// TIA Portal project "plc_industrial_sorter" (V17)

(* hardware
DEVICE "S7-1500/ET200MP station_1"  S7-1500 station
   slot 0: "Rail_0"  Rack  6ES7 590-1***0-0AA0
   slot 1: "PLC_1"  CPU 1511-1 PN  6ES7 511-1AK00-0AB0  V1.8
      slot 3: "CPU display_1"  6ES7591-1AA00-0AA0
      slot 32768: "PROFINET interface_1"  X1
         slot 32769: "Port_1"  X1 P1
         slot 32770: "Port_2"  X1 P2
*)

// ===== PLC "PLC_1"  CPU 1511-1 PN =====

DATA_BLOCK "Data_block_1"   // DB1
{ S7_Optimized_Access := 'TRUE' }
VERSION : 0.1
   VAR
      Nastro1_run : Bool;
      Fotocellula_ingresso_nastro1 : Bool;
      Val_induttivo : Bool;
      Val_capacitivo : Bool;
      Peso : Real;
      Fotocellula_scan : Bool;
      Fotocellula_ingresso_nastro2 : Bool;
      Tip_oggetto : Int := 0;
      Nastro2_run : Bool;
      Pusher_avanza : Bool;
      Pusher_rientra : Bool;
      Posizione_carrello : Int;
      State_machine : Int;
      Contenitore_target : Int;
      Posizione_target_carrello : Int;
      Posizione_oggetto_Y : Real;
      Posizione_oggetto_X : Real := -1000.0;
      Sistema_START : Bool;
      Sistema_STOP : Bool;
      Sistema_ANNULLA_ALLARMI : Bool;
      Sistema_avviato : Bool;
      tempvar1 : Int;
      Contatore : Int := -1;
      Allarme_generale : Bool;
   END_VAR
BEGIN
END_DATA_BLOCK

// folder: System blocks/Program resources

DATA_BLOCK "IEC_Timer_0_DB_2"   // DB4
{ S7_Optimized_Access := 'TRUE' }
AUTHOR : Simatic
FAMILY : IEC
NAME : IEC_TMR
VERSION : 1.0
// stored: InstanceOfName IEC_TIMER
"IEC_TIMER"
BEGIN
END_DATA_BLOCK

DATA_BLOCK "IEC_Timer_0_DB_1X"   // DB6
{ S7_Optimized_Access := 'TRUE' }
AUTHOR : Simatic
FAMILY : IEC
NAME : IEC_TMR
VERSION : 1.0
// stored: InstanceOfName IEC_TIMER
"IEC_TIMER"
BEGIN
END_DATA_BLOCK

DATA_BLOCK "IEC_Timer_0_DB_6"   // DB12
{ S7_Optimized_Access := 'TRUE' }
AUTHOR : Simatic
FAMILY : IEC
NAME : IEC_TMR
VERSION : 1.0
// stored: InstanceOfName IEC_TIMER
"IEC_TIMER"
BEGIN
END_DATA_BLOCK

DATA_BLOCK "IEC_Timer_0_DB_7"   // DB13
{ S7_Optimized_Access := 'TRUE' }
AUTHOR : Simatic
FAMILY : IEC
NAME : IEC_TMR
VERSION : 1.0
// stored: InstanceOfName IEC_TIMER
"IEC_TIMER"
BEGIN
END_DATA_BLOCK

DATA_BLOCK "IEC_Timer_0_DB_8"   // DB14
{ S7_Optimized_Access := 'TRUE' }
AUTHOR : Simatic
FAMILY : IEC
NAME : IEC_TMR
VERSION : 1.0
// stored: InstanceOfName IEC_TIMER
"IEC_TIMER"
BEGIN
END_DATA_BLOCK

DATA_BLOCK "IEC_Timer_0_DB_10"   // DB16
{ S7_Optimized_Access := 'TRUE' }
AUTHOR : Simatic
FAMILY : IEC
NAME : IEC_TMR
VERSION : 1.0
// stored: InstanceOfName IEC_TIMER
"IEC_TIMER"
BEGIN
END_DATA_BLOCK

DATA_BLOCK "IEC_Timer_0_DB_11"   // DB17
{ S7_Optimized_Access := 'TRUE' }
AUTHOR : Simatic
FAMILY : IEC
NAME : IEC_TMR
VERSION : 1.0
// stored: InstanceOfName IEC_TIMER
"IEC_TIMER"
BEGIN
END_DATA_BLOCK

DATA_BLOCK "IEC_Timer_0_DB_12"   // DB18
{ S7_Optimized_Access := 'TRUE' }
AUTHOR : Simatic
FAMILY : IEC
NAME : IEC_TMR
VERSION : 1.0
// stored: InstanceOfName IEC_TIMER
"IEC_TIMER"
BEGIN
END_DATA_BLOCK

// folder: (top level)

ORGANIZATION_BLOCK "Main"   // OB1, LAD, ProgramCycle
TITLE = "Main Program Sweep (Cycle)"
{ S7_Optimized_Access := 'TRUE' }
VERSION : 0.1
   VAR_INPUT
      Initial_Call : Bool;   // Initial call of this OB
      Remanence : Bool;   // =True, if remanent data are available
   END_VAR
   VAR_TEMP   // added for the SCL form of the ladder/FBD networks
      _w1 : Bool;
      _w2 : Bool;
   END_VAR
BEGIN

REGION Network 1
   // settato il blocco totale del sistema
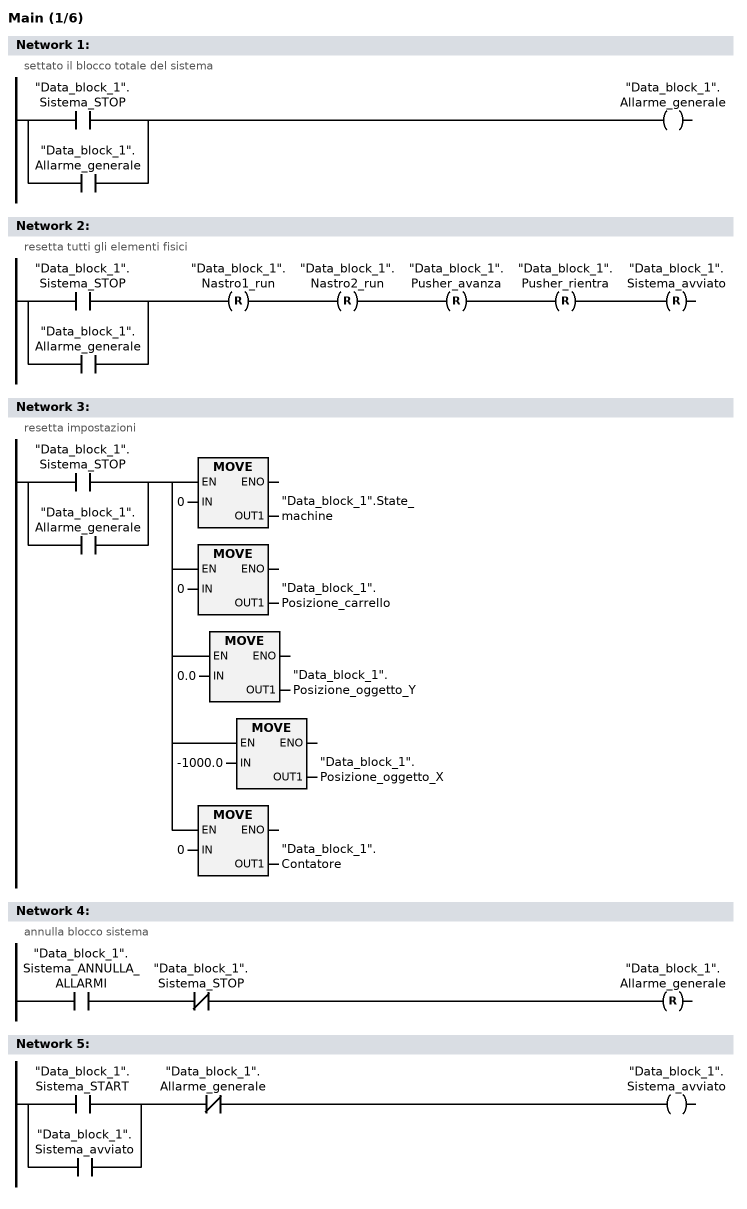
   RUNG wire#powerrail
      Contact( "Data_block_1".Sistema_STOP )
      wire#w1
      Coil( "Data_block_1".Allarme_generale )
   END_RUNG
   RUNG wire#powerrail
      Contact( "Data_block_1".Allarme_generale )
   END_RUNG wire#w1
   // the same network as SCL:
   "Data_block_1".Allarme_generale := "Data_block_1".Sistema_STOP OR "Data_block_1".Allarme_generale;
END_REGION

REGION Network 2
   // resetta tutti gli elementi fisici
   RUNG wire#powerrail
      Contact( "Data_block_1".Sistema_STOP )
      wire#w1
      R_Coil( "Data_block_1".Nastro1_run )
      R_Coil( "Data_block_1".Nastro2_run )
      R_Coil( "Data_block_1".Pusher_avanza )
      R_Coil( "Data_block_1".Pusher_rientra )
      R_Coil( "Data_block_1".Sistema_avviato )
   END_RUNG
   RUNG wire#powerrail
      Contact( "Data_block_1".Allarme_generale )
   END_RUNG wire#w1
   // the same network as SCL:
   IF "Data_block_1".Sistema_STOP OR "Data_block_1".Allarme_generale THEN
       "Data_block_1".Nastro1_run := FALSE;
       "Data_block_1".Nastro2_run := FALSE;
       "Data_block_1".Pusher_avanza := FALSE;
       "Data_block_1".Pusher_rientra := FALSE;
       "Data_block_1".Sistema_avviato := FALSE;
   END_IF;
END_REGION

REGION Network 3
   // resetta impostazioni
   RUNG wire#powerrail
      Contact( "Data_block_1".Sistema_STOP )
      wire#w1
      Move(in := 0, out1 => "Data_block_1".State_machine)
   END_RUNG
   RUNG wire#powerrail
      Contact( "Data_block_1".Allarme_generale )
   END_RUNG wire#w1
   RUNG wire#w1
      Move(in := 0, out1 => "Data_block_1".Posizione_carrello)
   END_RUNG
   RUNG wire#w1
      Move(in := 0.0, out1 => "Data_block_1".Posizione_oggetto_Y)
   END_RUNG
   RUNG wire#w1
      Move(in := -1000.0, out1 => "Data_block_1".Posizione_oggetto_X)
   END_RUNG
   RUNG wire#w1
      Move(in := 0, out1 => "Data_block_1".Contatore)
   END_RUNG
   // the same network as SCL:
   IF "Data_block_1".Sistema_STOP OR "Data_block_1".Allarme_generale THEN
       "Data_block_1".State_machine := 0;
       "Data_block_1".Posizione_carrello := 0;
       "Data_block_1".Posizione_oggetto_Y := 0.0;
       "Data_block_1".Posizione_oggetto_X := -1000.0;
       "Data_block_1".Contatore := 0;
   END_IF;
END_REGION

REGION Network 4
   // annulla blocco sistema
   RUNG wire#powerrail
      Contact( "Data_block_1".Sistema_ANNULLA_ALLARMI )
      I_Contact( "Data_block_1".Sistema_STOP )
      R_Coil( "Data_block_1".Allarme_generale )
   END_RUNG
   // the same network as SCL:
   IF "Data_block_1".Sistema_ANNULLA_ALLARMI AND NOT "Data_block_1".Sistema_STOP THEN
       "Data_block_1".Allarme_generale := FALSE;
   END_IF;
END_REGION

REGION Network 5
   RUNG wire#powerrail
      Contact( "Data_block_1".Sistema_START )
      wire#w1
      I_Contact( "Data_block_1".Allarme_generale )
      Coil( "Data_block_1".Sistema_avviato )
   END_RUNG
   RUNG wire#powerrail
      Contact( "Data_block_1".Sistema_avviato )
   END_RUNG wire#w1
   // the same network as SCL:
   "Data_block_1".Sistema_avviato := ("Data_block_1".Sistema_START OR "Data_block_1".Sistema_avviato) AND NOT "Data_block_1".Allarme_generale;
END_REGION

REGION Network 6
   // rung supporto (inizializza la fotocellula primo avvio)
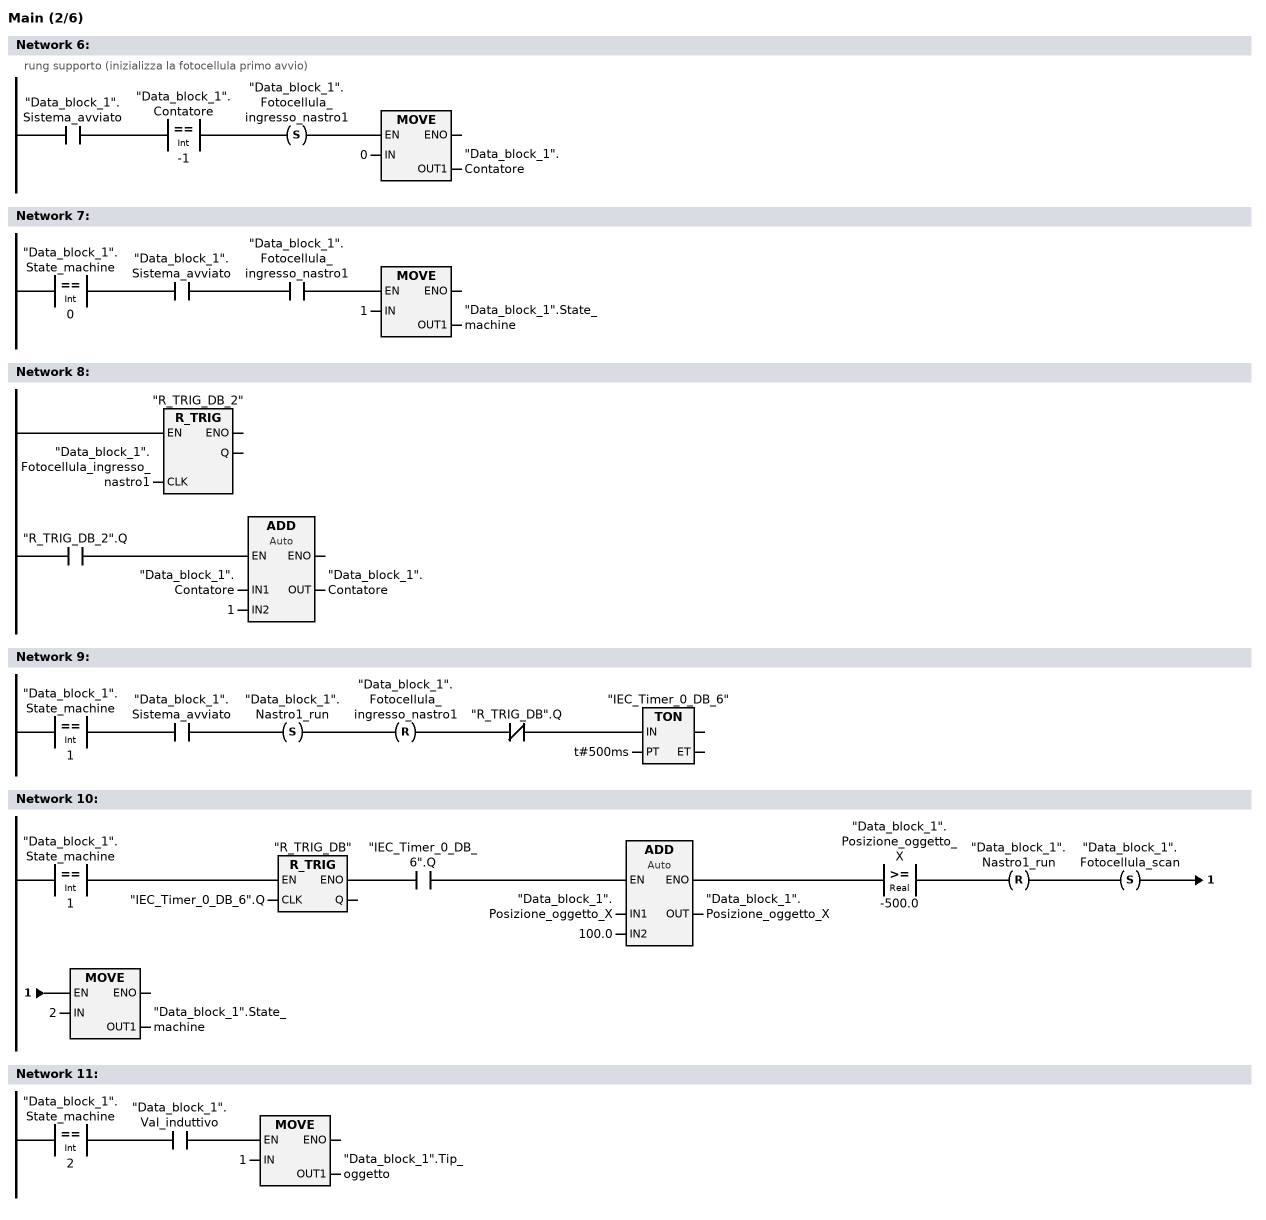
   RUNG wire#powerrail
      Contact( "Data_block_1".Sistema_avviato )
      { S7_Templates := "SrcType := Int" } EQ_Contact(in1 := "Data_block_1".Contatore, in2 := -1)
      S_Coil( "Data_block_1".Fotocellula_ingresso_nastro1 )
      Move(in := 0, out1 => "Data_block_1".Contatore)
   END_RUNG
   // the same network as SCL:
   IF "Data_block_1".Sistema_avviato AND ("Data_block_1".Contatore = (-1)) THEN
       "Data_block_1".Fotocellula_ingresso_nastro1 := TRUE;
       "Data_block_1".Contatore := 0;
   END_IF;
END_REGION

REGION Network 7
   RUNG wire#powerrail
      { S7_Templates := "SrcType := Int" } EQ_Contact(in1 := "Data_block_1".State_machine, in2 := 0)
      Contact( "Data_block_1".Sistema_avviato )
      Contact( "Data_block_1".Fotocellula_ingresso_nastro1 )
      Move(in := 1, out1 => "Data_block_1".State_machine)
   END_RUNG
   // the same network as SCL:
   IF ("Data_block_1".State_machine = 0) AND "Data_block_1".Sistema_avviato AND "Data_block_1".Fotocellula_ingresso_nastro1 THEN
       "Data_block_1".State_machine := 1;
   END_IF;
END_REGION

REGION Network 8
   "R_TRIG_DB_2"(CLK := "Data_block_1".Fotocellula_ingresso_nastro1);   // R_TRIG
   IF "R_TRIG_DB_2".Q THEN "Data_block_1".Contatore := "Data_block_1".Contatore + 1; END_IF;
END_REGION

REGION Network 9
   #_w1 := ("Data_block_1".State_machine = 1) AND "Data_block_1".Sistema_avviato;
   IF #_w1 THEN
       "Data_block_1".Nastro1_run := TRUE;
       "Data_block_1".Fotocellula_ingresso_nastro1 := FALSE;
   END_IF;
   "IEC_Timer_0_DB_6".TON(IN := #_w1 AND NOT "R_TRIG_DB".Q, PT := t#500ms);
END_REGION

REGION Network 10
   // ENO of a box is taken as its EN; it also drops when the box reports an error
   #_w1 := "Data_block_1".State_machine = 1;
   IF #_w1 THEN
       "R_TRIG_DB"(CLK := "IEC_Timer_0_DB_6".Q);   // R_TRIG
   END_IF;
   #_w2 := #_w1 AND "IEC_Timer_0_DB_6".Q;
   IF #_w2 THEN "Data_block_1".Posizione_oggetto_X := "Data_block_1".Posizione_oggetto_X + 100.0; END_IF;
   IF #_w2 AND ("Data_block_1".Posizione_oggetto_X >= (-500.0)) THEN
       "Data_block_1".Nastro1_run := FALSE;
       "Data_block_1".Fotocellula_scan := TRUE;
       "Data_block_1".State_machine := 2;
   END_IF;
END_REGION

REGION Network 11
   RUNG wire#powerrail
      { S7_Templates := "SrcType := Int" } EQ_Contact(in1 := "Data_block_1".State_machine, in2 := 2)
      Contact( "Data_block_1".Val_induttivo )
      Move(in := 1, out1 => "Data_block_1".Tip_oggetto)
   END_RUNG
   // the same network as SCL:
   IF ("Data_block_1".State_machine = 2) AND "Data_block_1".Val_induttivo THEN
       "Data_block_1".Tip_oggetto := 1;
   END_IF;
END_REGION

REGION Network 12
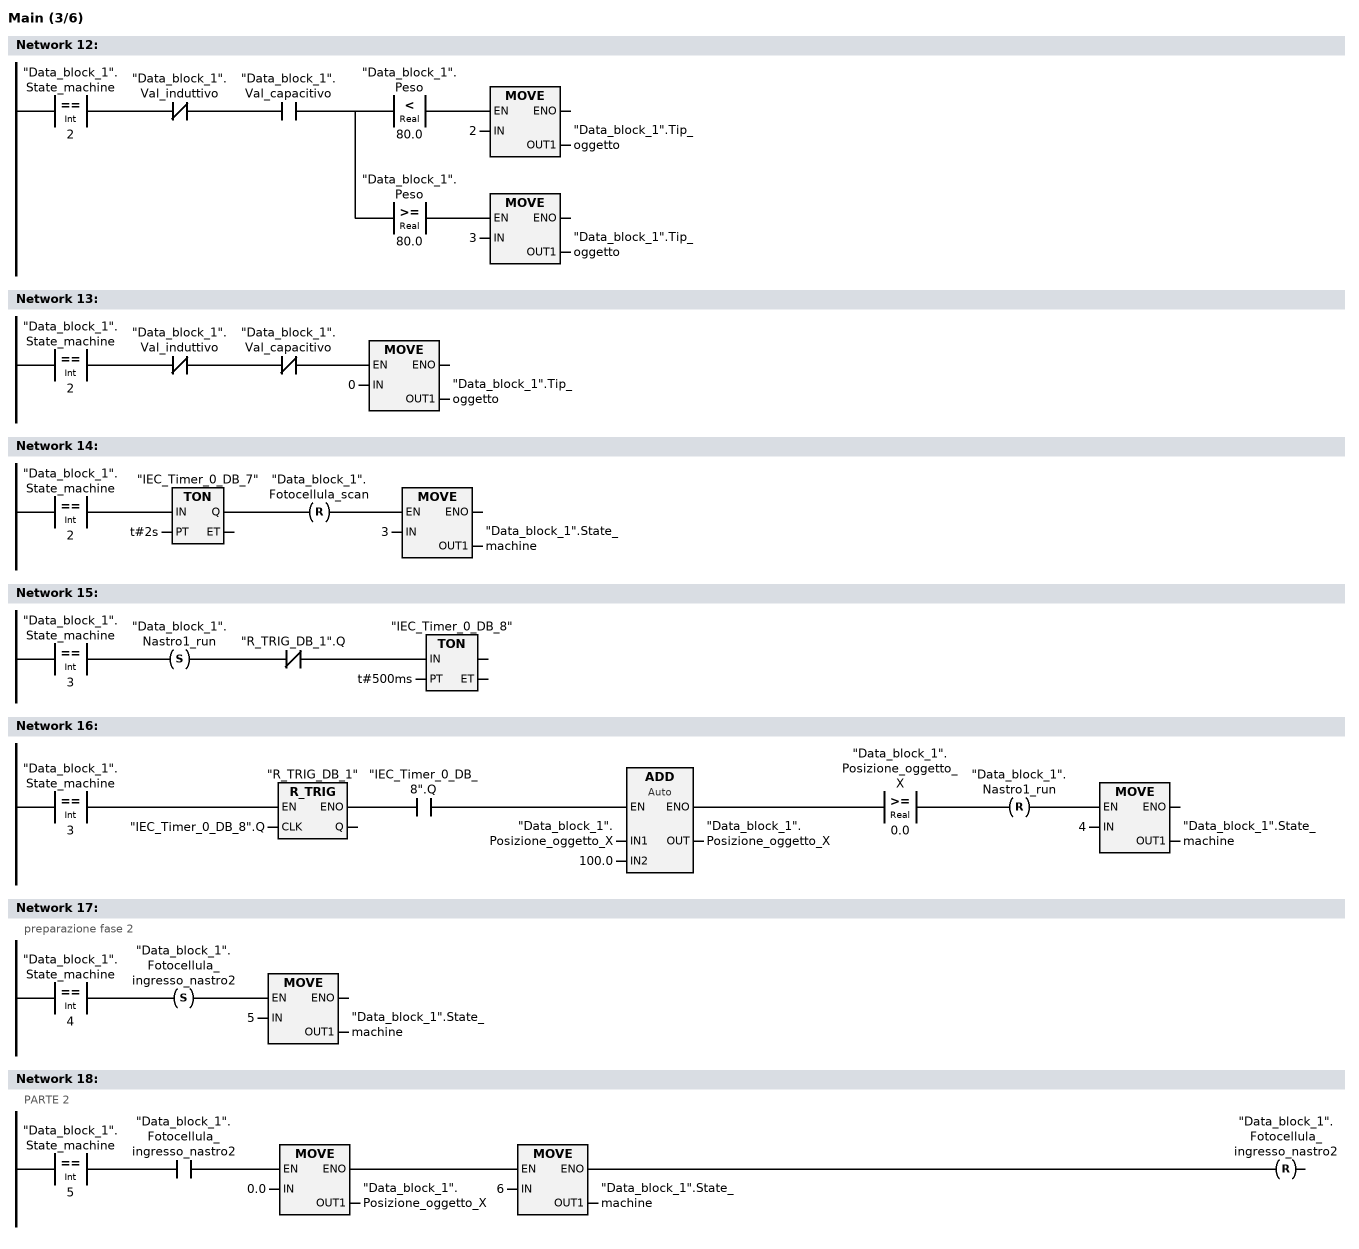
   RUNG wire#powerrail
      { S7_Templates := "SrcType := Int" } EQ_Contact(in1 := "Data_block_1".State_machine, in2 := 2)
      I_Contact( "Data_block_1".Val_induttivo )
      Contact( "Data_block_1".Val_capacitivo )
      wire#w1
      { S7_Templates := "SrcType := Real" } LT_Contact(in1 := "Data_block_1".Peso, in2 := 80.0)
      Move(in := 2, out1 => "Data_block_1".Tip_oggetto)
   END_RUNG
   RUNG wire#w1
      { S7_Templates := "SrcType := Real" } GE_Contact(in1 := "Data_block_1".Peso, in2 := 80.0)
      Move(in := 3, out1 => "Data_block_1".Tip_oggetto)
   END_RUNG
   // the same network as SCL:
   #_w1 := ("Data_block_1".State_machine = 2) AND NOT "Data_block_1".Val_induttivo AND "Data_block_1".Val_capacitivo;
   IF #_w1 AND ("Data_block_1".Peso < 80.0) THEN "Data_block_1".Tip_oggetto := 2; END_IF;
   IF #_w1 AND ("Data_block_1".Peso >= 80.0) THEN "Data_block_1".Tip_oggetto := 3; END_IF;
END_REGION

REGION Network 13
   RUNG wire#powerrail
      { S7_Templates := "SrcType := Int" } EQ_Contact(in1 := "Data_block_1".State_machine, in2 := 2)
      I_Contact( "Data_block_1".Val_induttivo )
      I_Contact( "Data_block_1".Val_capacitivo )
      Move(in := 0, out1 => "Data_block_1".Tip_oggetto)
   END_RUNG
   // the same network as SCL:
   IF ("Data_block_1".State_machine = 2) AND NOT "Data_block_1".Val_induttivo AND NOT "Data_block_1".Val_capacitivo THEN
       "Data_block_1".Tip_oggetto := 0;
   END_IF;
END_REGION

REGION Network 14
   "IEC_Timer_0_DB_7".TON(IN := "Data_block_1".State_machine = 2, PT := t#2s);
   IF "IEC_Timer_0_DB_7".Q THEN
       "Data_block_1".Fotocellula_scan := FALSE;
       "Data_block_1".State_machine := 3;
   END_IF;
END_REGION

REGION Network 15
   #_w1 := "Data_block_1".State_machine = 3;
   IF #_w1 THEN "Data_block_1".Nastro1_run := TRUE; END_IF;
   "IEC_Timer_0_DB_8".TON(IN := #_w1 AND NOT "R_TRIG_DB_1".Q, PT := t#500ms);
END_REGION

REGION Network 16
   // ENO of a box is taken as its EN; it also drops when the box reports an error
   #_w1 := "Data_block_1".State_machine = 3;
   IF #_w1 THEN
       "R_TRIG_DB_1"(CLK := "IEC_Timer_0_DB_8".Q);   // R_TRIG
   END_IF;
   #_w2 := #_w1 AND "IEC_Timer_0_DB_8".Q;
   IF #_w2 THEN "Data_block_1".Posizione_oggetto_X := "Data_block_1".Posizione_oggetto_X + 100.0; END_IF;
   IF #_w2 AND ("Data_block_1".Posizione_oggetto_X >= 0.0) THEN
       "Data_block_1".Nastro1_run := FALSE;
       "Data_block_1".State_machine := 4;
   END_IF;
END_REGION

REGION Network 17
   // preparazione fase 2
   RUNG wire#powerrail
      { S7_Templates := "SrcType := Int" } EQ_Contact(in1 := "Data_block_1".State_machine, in2 := 4)
      S_Coil( "Data_block_1".Fotocellula_ingresso_nastro2 )
      Move(in := 5, out1 => "Data_block_1".State_machine)
   END_RUNG
   // the same network as SCL:
   IF "Data_block_1".State_machine = 4 THEN
       "Data_block_1".Fotocellula_ingresso_nastro2 := TRUE;
       "Data_block_1".State_machine := 5;
   END_IF;
END_REGION

REGION Network 18
   // PARTE 2
   RUNG wire#powerrail
      { S7_Templates := "SrcType := Int" } EQ_Contact(in1 := "Data_block_1".State_machine, in2 := 5)
      Contact( "Data_block_1".Fotocellula_ingresso_nastro2 )
      Move(in := 0.0, out1 => "Data_block_1".Posizione_oggetto_X)
      Move(in := 6, out1 => "Data_block_1".State_machine)
      R_Coil( "Data_block_1".Fotocellula_ingresso_nastro2 )
   END_RUNG
   // the same network as SCL:
   IF ("Data_block_1".State_machine = 5) AND "Data_block_1".Fotocellula_ingresso_nastro2 THEN
       "Data_block_1".Posizione_oggetto_X := 0.0;
   END_IF;
   #_w1 := ("Data_block_1".State_machine = 5) AND "Data_block_1".Fotocellula_ingresso_nastro2;
   IF #_w1 THEN
       "Data_block_1".State_machine := 6;
       "Data_block_1".Fotocellula_ingresso_nastro2 := FALSE;
   END_IF;
END_REGION

REGION Network 19
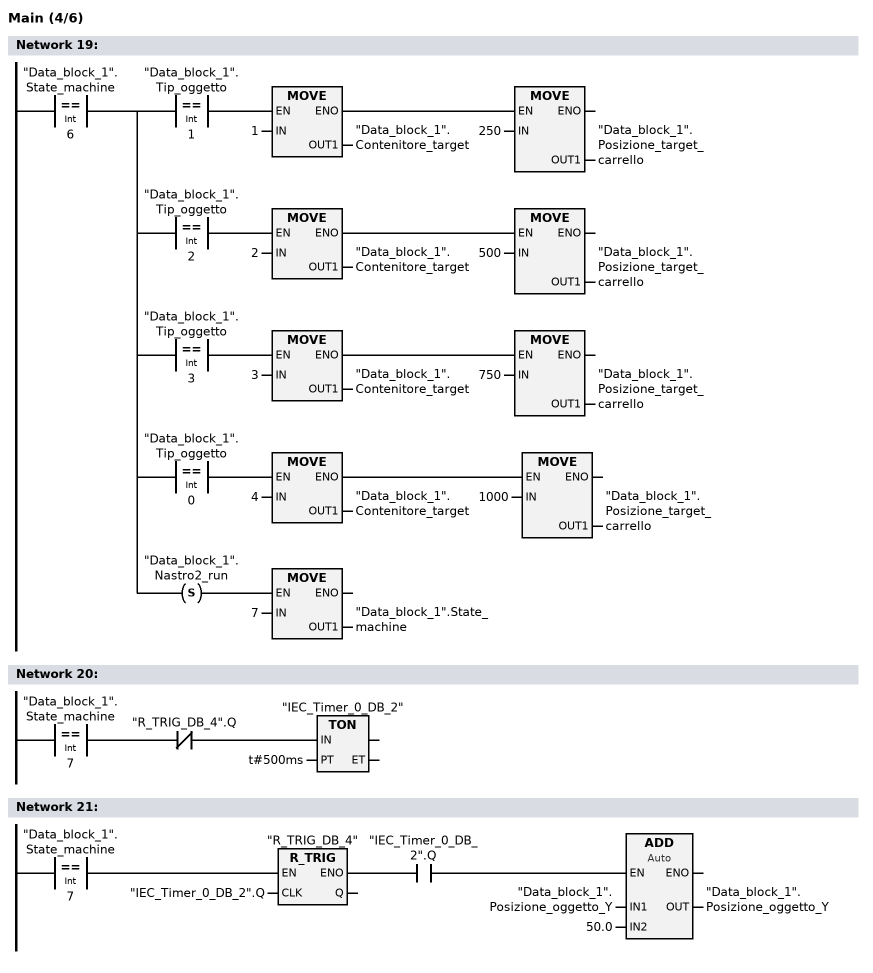
   RUNG wire#powerrail
      { S7_Templates := "SrcType := Int" } EQ_Contact(in1 := "Data_block_1".State_machine, in2 := 6)
      wire#w1
      { S7_Templates := "SrcType := Int" } EQ_Contact(in1 := "Data_block_1".Tip_oggetto, in2 := 1)
      Move(in := 1, out1 => "Data_block_1".Contenitore_target)
      Move(in := 250, out1 => "Data_block_1".Posizione_target_carrello)
   END_RUNG
   RUNG wire#w1
      { S7_Templates := "SrcType := Int" } EQ_Contact(in1 := "Data_block_1".Tip_oggetto, in2 := 2)
      Move(in := 2, out1 => "Data_block_1".Contenitore_target)
      Move(in := 500, out1 => "Data_block_1".Posizione_target_carrello)
   END_RUNG
   RUNG wire#w1
      { S7_Templates := "SrcType := Int" } EQ_Contact(in1 := "Data_block_1".Tip_oggetto, in2 := 3)
      Move(in := 3, out1 => "Data_block_1".Contenitore_target)
      Move(in := 750, out1 => "Data_block_1".Posizione_target_carrello)
   END_RUNG
   RUNG wire#w1
      { S7_Templates := "SrcType := Int" } EQ_Contact(in1 := "Data_block_1".Tip_oggetto, in2 := 0)
      Move(in := 4, out1 => "Data_block_1".Contenitore_target)
      Move(in := 1000, out1 => "Data_block_1".Posizione_target_carrello)
   END_RUNG
   RUNG wire#w1
      S_Coil( "Data_block_1".Nastro2_run )
      Move(in := 7, out1 => "Data_block_1".State_machine)
   END_RUNG
   // the same network as SCL:
   #_w1 := "Data_block_1".State_machine = 6;
   IF #_w1 AND ("Data_block_1".Tip_oggetto = 1) THEN
       "Data_block_1".Contenitore_target := 1;
       "Data_block_1".Posizione_target_carrello := 250;
   END_IF;
   IF #_w1 AND ("Data_block_1".Tip_oggetto = 2) THEN
       "Data_block_1".Contenitore_target := 2;
       "Data_block_1".Posizione_target_carrello := 500;
   END_IF;
   IF #_w1 AND ("Data_block_1".Tip_oggetto = 3) THEN
       "Data_block_1".Contenitore_target := 3;
       "Data_block_1".Posizione_target_carrello := 750;
   END_IF;
   IF #_w1 AND ("Data_block_1".Tip_oggetto = 0) THEN
       "Data_block_1".Contenitore_target := 4;
       "Data_block_1".Posizione_target_carrello := 1000;
   END_IF;
   IF #_w1 THEN
       "Data_block_1".Nastro2_run := TRUE;
       "Data_block_1".State_machine := 7;
   END_IF;
END_REGION

REGION Network 20
   "IEC_Timer_0_DB_2".TON(IN := ("Data_block_1".State_machine = 7) AND NOT "R_TRIG_DB_4".Q, PT := t#500ms);
END_REGION

REGION Network 21
   // ENO of a box is taken as its EN; it also drops when the box reports an error
   #_w1 := "Data_block_1".State_machine = 7;
   IF #_w1 THEN
       "R_TRIG_DB_4"(CLK := "IEC_Timer_0_DB_2".Q);   // R_TRIG
   END_IF;
   IF #_w1 AND "IEC_Timer_0_DB_2".Q THEN
       "Data_block_1".Posizione_oggetto_Y := "Data_block_1".Posizione_oggetto_Y + 50.0;
   END_IF;
END_REGION

REGION Network 22
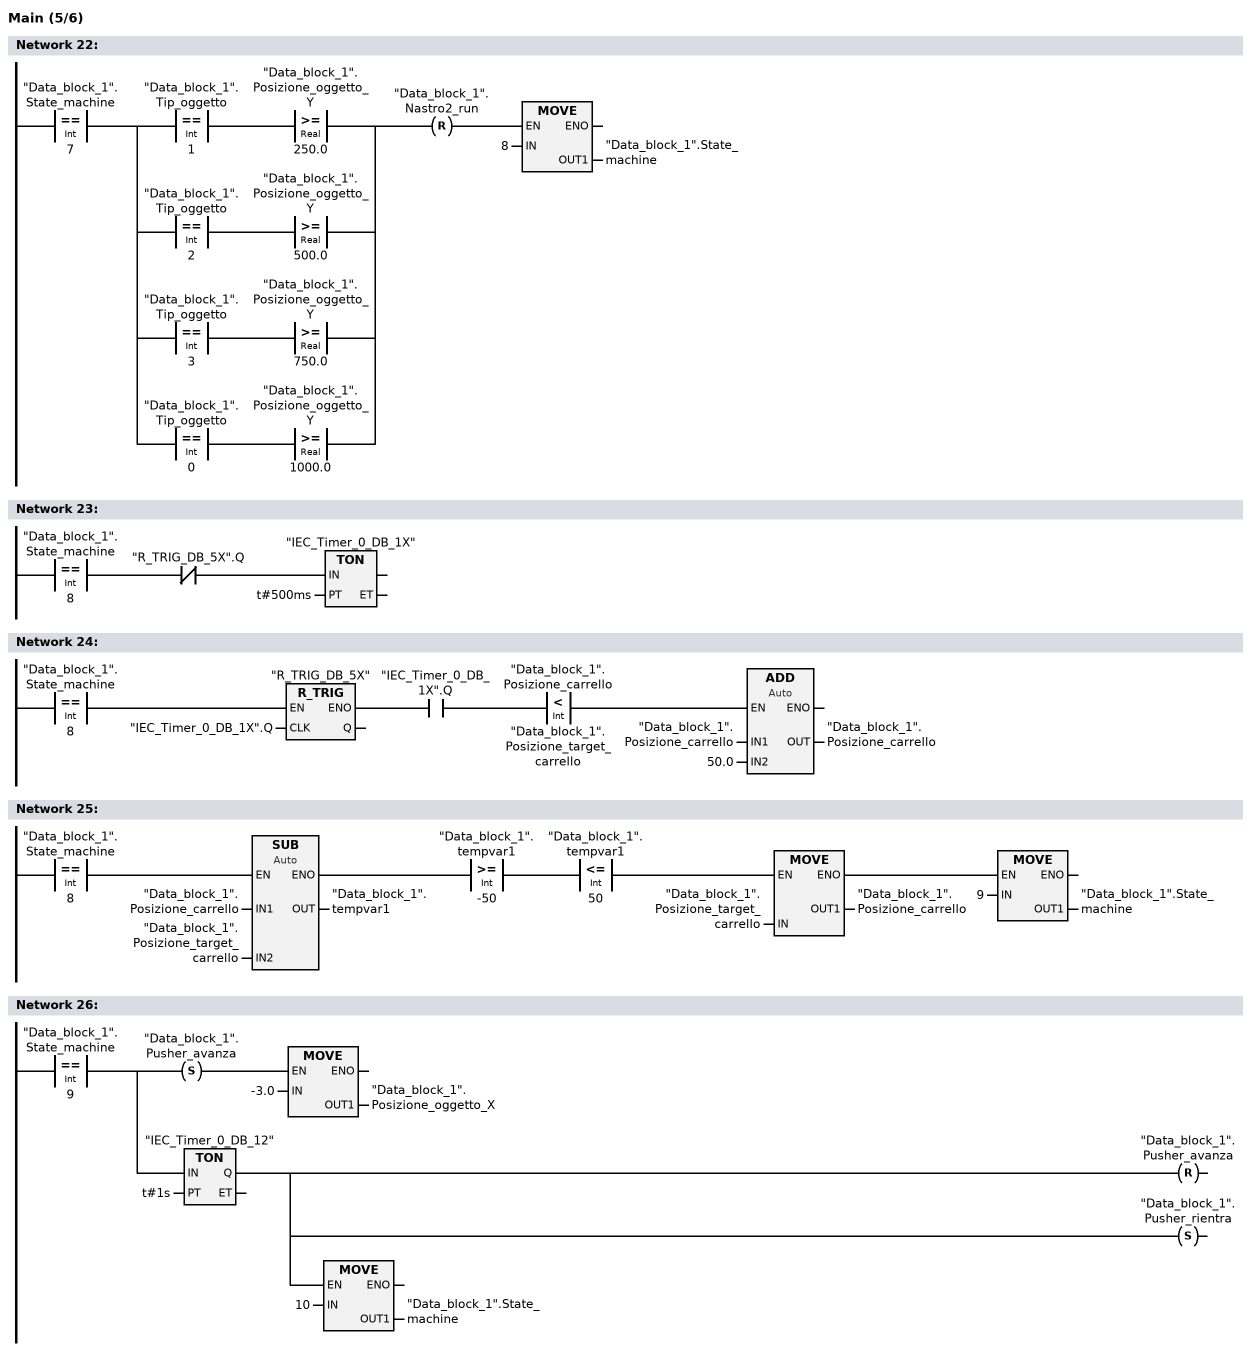
   RUNG wire#powerrail
      { S7_Templates := "SrcType := Int" } EQ_Contact(in1 := "Data_block_1".State_machine, in2 := 7)
      wire#w1
      { S7_Templates := "SrcType := Int" } EQ_Contact(in1 := "Data_block_1".Tip_oggetto, in2 := 1)
      { S7_Templates := "SrcType := Real" } GE_Contact(in1 := "Data_block_1".Posizione_oggetto_Y, in2 := 250.0)
      wire#w2
      R_Coil( "Data_block_1".Nastro2_run )
      Move(in := 8, out1 => "Data_block_1".State_machine)
   END_RUNG
   RUNG wire#w1
      { S7_Templates := "SrcType := Int" } EQ_Contact(in1 := "Data_block_1".Tip_oggetto, in2 := 2)
      { S7_Templates := "SrcType := Real" } GE_Contact(in1 := "Data_block_1".Posizione_oggetto_Y, in2 := 500.0)
   END_RUNG wire#w2
   RUNG wire#w1
      { S7_Templates := "SrcType := Int" } EQ_Contact(in1 := "Data_block_1".Tip_oggetto, in2 := 3)
      { S7_Templates := "SrcType := Real" } GE_Contact(in1 := "Data_block_1".Posizione_oggetto_Y, in2 := 750.0)
   END_RUNG wire#w2
   RUNG wire#w1
      { S7_Templates := "SrcType := Int" } EQ_Contact(in1 := "Data_block_1".Tip_oggetto, in2 := 0)
      { S7_Templates := "SrcType := Real" } GE_Contact(in1 := "Data_block_1".Posizione_oggetto_Y, in2 := 1000.0)
   END_RUNG wire#w2
   // the same network as SCL:
   IF ("Data_block_1".State_machine = 7) AND ((("Data_block_1".Tip_oggetto = 1) AND ("Data_block_1".Posizione_oggetto_Y >= 250.0)) OR (("Data_block_1".Tip_oggetto = 2) AND ("Data_block_1".Posizione_oggetto_Y >= 500.0)) OR (("Data_block_1".Tip_oggetto = 3) AND ("Data_block_1".Posizione_oggetto_Y >= 750.0)) OR (("Data_block_1".Tip_oggetto = 0) AND ("Data_block_1".Posizione_oggetto_Y >= 1000.0))) THEN
       "Data_block_1".Nastro2_run := FALSE;
       "Data_block_1".State_machine := 8;
   END_IF;
END_REGION

REGION Network 23
   "IEC_Timer_0_DB_1X".TON(IN := ("Data_block_1".State_machine = 8) AND NOT "R_TRIG_DB_5X".Q, PT := t#500ms);
END_REGION

REGION Network 24
   // ENO of a box is taken as its EN; it also drops when the box reports an error
   #_w1 := "Data_block_1".State_machine = 8;
   IF #_w1 THEN
       "R_TRIG_DB_5X"(CLK := "IEC_Timer_0_DB_1X".Q);   // R_TRIG
   END_IF;
   IF #_w1 AND "IEC_Timer_0_DB_1X".Q AND ("Data_block_1".Posizione_carrello < "Data_block_1".Posizione_target_carrello) THEN
       "Data_block_1".Posizione_carrello := "Data_block_1".Posizione_carrello + 50.0;
   END_IF;
END_REGION

REGION Network 25
   RUNG wire#powerrail
      { S7_Templates := "SrcType := Int" } EQ_Contact(in1 := "Data_block_1".State_machine, in2 := 8)
      Sub(in1 := "Data_block_1".Posizione_carrello, in2 := "Data_block_1".Posizione_target_carrello, out => "Data_block_1".tempvar1)
      { S7_Templates := "SrcType := Int" } GE_Contact(in1 := "Data_block_1".tempvar1, in2 := -50)
      { S7_Templates := "SrcType := Int" } LE_Contact(in1 := "Data_block_1".tempvar1, in2 := 50)
      Move(in := "Data_block_1".Posizione_target_carrello, out1 => "Data_block_1".Posizione_carrello)
      Move(in := 9, out1 => "Data_block_1".State_machine)
   END_RUNG
   // the same network as SCL:
   #_w1 := "Data_block_1".State_machine = 8;
   IF #_w1 THEN
       "Data_block_1".tempvar1 := "Data_block_1".Posizione_carrello - "Data_block_1".Posizione_target_carrello;
   END_IF;
   IF #_w1 AND ("Data_block_1".tempvar1 >= (-50)) AND ("Data_block_1".tempvar1 <= 50) THEN
       "Data_block_1".Posizione_carrello := "Data_block_1".Posizione_target_carrello;
       "Data_block_1".State_machine := 9;
   END_IF;
END_REGION

REGION Network 26
   #_w1 := "Data_block_1".State_machine = 9;
   IF #_w1 THEN
       "Data_block_1".Pusher_avanza := TRUE;
       "Data_block_1".Posizione_oggetto_X := -3.0;
   END_IF;
   "IEC_Timer_0_DB_12".TON(IN := #_w1, PT := t#1s);
   IF "IEC_Timer_0_DB_12".Q THEN
       "Data_block_1".Pusher_avanza := FALSE;
       "Data_block_1".Pusher_rientra := TRUE;
       "Data_block_1".State_machine := 10;
   END_IF;
END_REGION

REGION Network 27
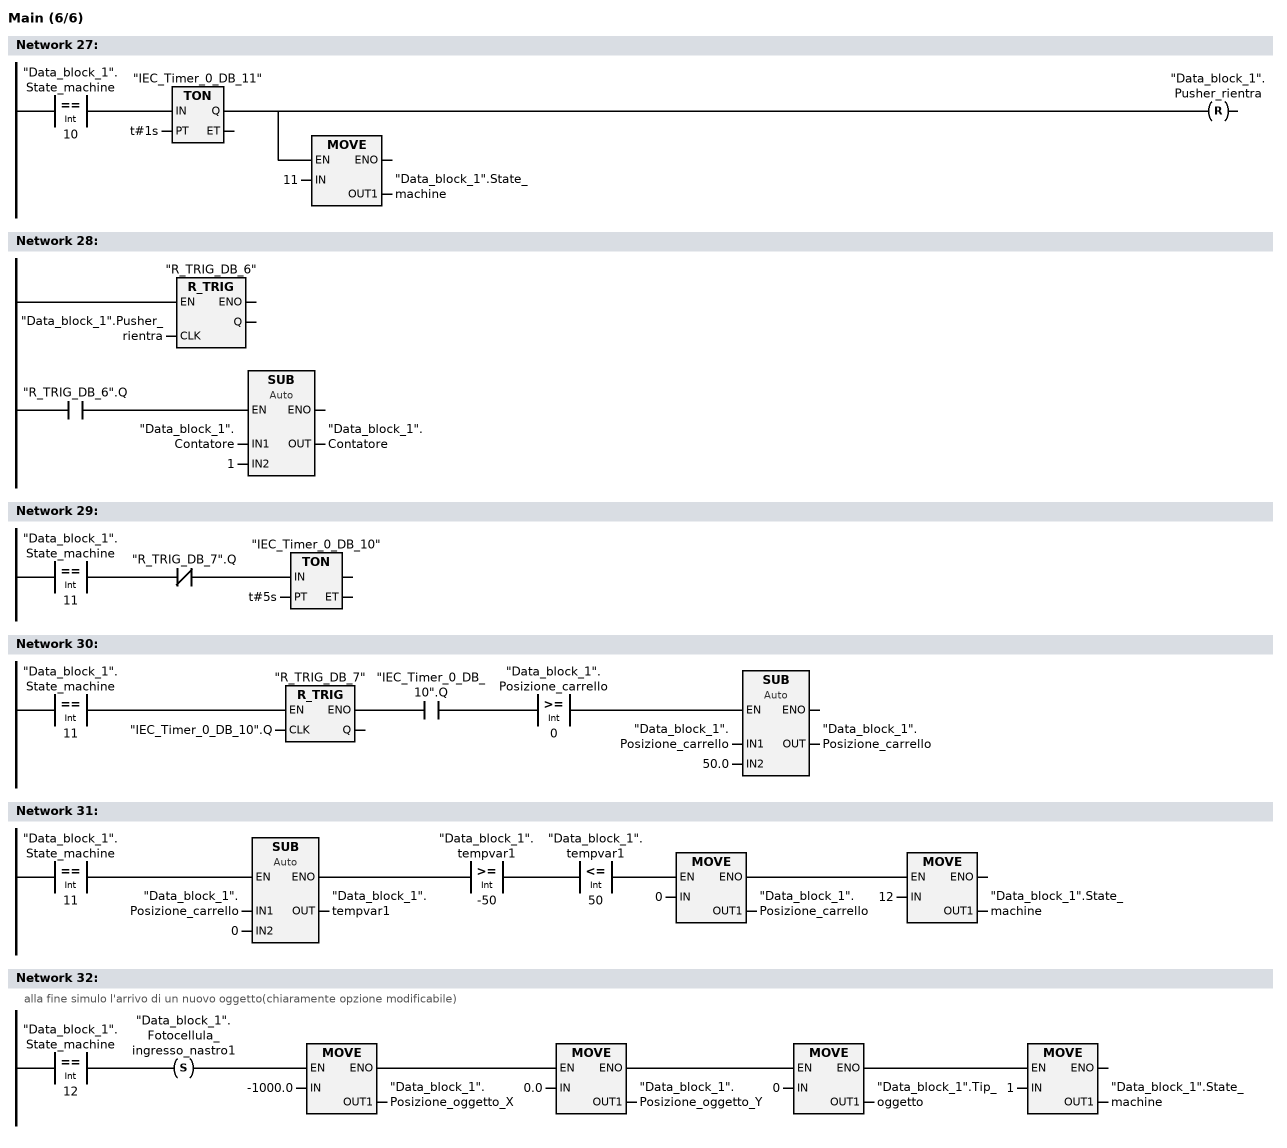
   "IEC_Timer_0_DB_11".TON(IN := "Data_block_1".State_machine = 10, PT := t#1s);
   IF "IEC_Timer_0_DB_11".Q THEN
       "Data_block_1".Pusher_rientra := FALSE;
       "Data_block_1".State_machine := 11;
   END_IF;
END_REGION

REGION Network 28
   "R_TRIG_DB_6"(CLK := "Data_block_1".Pusher_rientra);   // R_TRIG
   IF "R_TRIG_DB_6".Q THEN "Data_block_1".Contatore := "Data_block_1".Contatore - 1; END_IF;
END_REGION

REGION Network 29
   "IEC_Timer_0_DB_10".TON(IN := ("Data_block_1".State_machine = 11) AND NOT "R_TRIG_DB_7".Q, PT := t#5s);
END_REGION

REGION Network 30
   // ENO of a box is taken as its EN; it also drops when the box reports an error
   #_w1 := "Data_block_1".State_machine = 11;
   IF #_w1 THEN
       "R_TRIG_DB_7"(CLK := "IEC_Timer_0_DB_10".Q);   // R_TRIG
   END_IF;
   IF #_w1 AND "IEC_Timer_0_DB_10".Q AND ("Data_block_1".Posizione_carrello >= 0) THEN
       "Data_block_1".Posizione_carrello := "Data_block_1".Posizione_carrello - 50.0;
   END_IF;
END_REGION

REGION Network 31
   RUNG wire#powerrail
      { S7_Templates := "SrcType := Int" } EQ_Contact(in1 := "Data_block_1".State_machine, in2 := 11)
      Sub(in1 := "Data_block_1".Posizione_carrello, in2 := 0, out => "Data_block_1".tempvar1)
      { S7_Templates := "SrcType := Int" } GE_Contact(in1 := "Data_block_1".tempvar1, in2 := -50)
      { S7_Templates := "SrcType := Int" } LE_Contact(in1 := "Data_block_1".tempvar1, in2 := 50)
      Move(in := 0, out1 => "Data_block_1".Posizione_carrello)
      Move(in := 12, out1 => "Data_block_1".State_machine)
   END_RUNG
   // the same network as SCL:
   #_w1 := "Data_block_1".State_machine = 11;
   IF #_w1 THEN "Data_block_1".tempvar1 := "Data_block_1".Posizione_carrello - 0; END_IF;
   IF #_w1 AND ("Data_block_1".tempvar1 >= (-50)) AND ("Data_block_1".tempvar1 <= 50) THEN
       "Data_block_1".Posizione_carrello := 0;
       "Data_block_1".State_machine := 12;
   END_IF;
END_REGION

REGION Network 32
   // alla fine simulo l'arrivo di un nuovo oggetto(chiaramente opzione modificabile)
   RUNG wire#powerrail
      { S7_Templates := "SrcType := Int" } EQ_Contact(in1 := "Data_block_1".State_machine, in2 := 12)
      S_Coil( "Data_block_1".Fotocellula_ingresso_nastro1 )
      Move(in := -1000.0, out1 => "Data_block_1".Posizione_oggetto_X)
      Move(in := 0.0, out1 => "Data_block_1".Posizione_oggetto_Y)
      Move(in := 0, out1 => "Data_block_1".Tip_oggetto)
      Move(in := 1, out1 => "Data_block_1".State_machine)
   END_RUNG
   // the same network as SCL:
   IF "Data_block_1".State_machine = 12 THEN
       "Data_block_1".Fotocellula_ingresso_nastro1 := TRUE;
       "Data_block_1".Posizione_oggetto_X := -1000.0;
       "Data_block_1".Posizione_oggetto_Y := 0.0;
       "Data_block_1".Tip_oggetto := 0;
       "Data_block_1".State_machine := 1;
   END_IF;
END_REGION
END_ORGANIZATION_BLOCK